{attribute 'GeneratedUsingTerminal: EK1122-0000-0018'}
{attribute addProperty BoxType "EK1122-0000-0018"}
{attribute addProperty Id "Beckhoff_AMI8xxxsub_EK1100EK1100_AB5A94672A_0001_AMI8000_0000_0016AMI8000_A36814CB39A_0002_AMI8000_0090_0016AMI8000_A36814CB39"}
{attribute addProperty CRC "3966058734"}
{attribute addProperty Size "80"}
TYPE Beckhoff_AMI8xxxEK1122_EC6540EE EXTENDS EK1122_AB5A9467 :
STRUCT
	{attribute addProperty Name "Beckhoff_AMI8xxxsub_EK1100"}
	Beckhoff_AMI8xxxsub_EK1100 : EK1100_AB5A9467;
	{attribute addProperty Name "A_0001_AMI8000_0000_0016"}
	A_0001_AMI8000_0000_0016 : AMI8000_A36814CB;
	{attribute addProperty Name "A_0002_AMI8000_0090_0016"}
	A_0002_AMI8000_0090_0016 : AMI8000_A36814CB;
END_STRUCT
END_TYPE

(* stored: Version 1.2.0.0, ProductVersion 3.1.4024.9
   DUT Beckhoff_AMI8xxxEK1122_EC6540EE: Id {c1f2afd3-5ccb-4650-9f89-2c1339c94cea} *)
